FUNCTION_BLOCK FB_WATCHDOG_T (* Enables watchdog timeouts longer than the default. *)
  (* Standard: 61499-2; Description: TIMEOUT must be less than 15 s. The lower DT, the more accurate, but the higher the internal clock rate. *)
  (* Version 1.0, 2017-09-12, Marc Jakobi, HTW Berlin *)
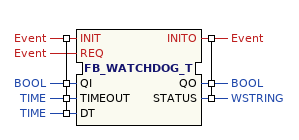
  EVENT_INPUT
    INIT WITH QI, TIMEOUT, DT; (* Initialization Request *)
    REQ; (* Normal Execution Request *)
  END_EVENT
  EVENT_OUTPUT
    INITO WITH QO, STATUS; (* Initialization Confirm *)
  END_EVENT
  VAR_INPUT
    QI : BOOL; (* Input event qualifier *)
    TIMEOUT : TIME; (* Watchdog timeout *)
    DT : TIME; (* Watchdog pet interval *)
  END_VAR
  VAR_OUTPUT
    QO : BOOL; (* Output event qualifier *)
    STATUS : WSTRING; (* Service status *)
  END_VAR
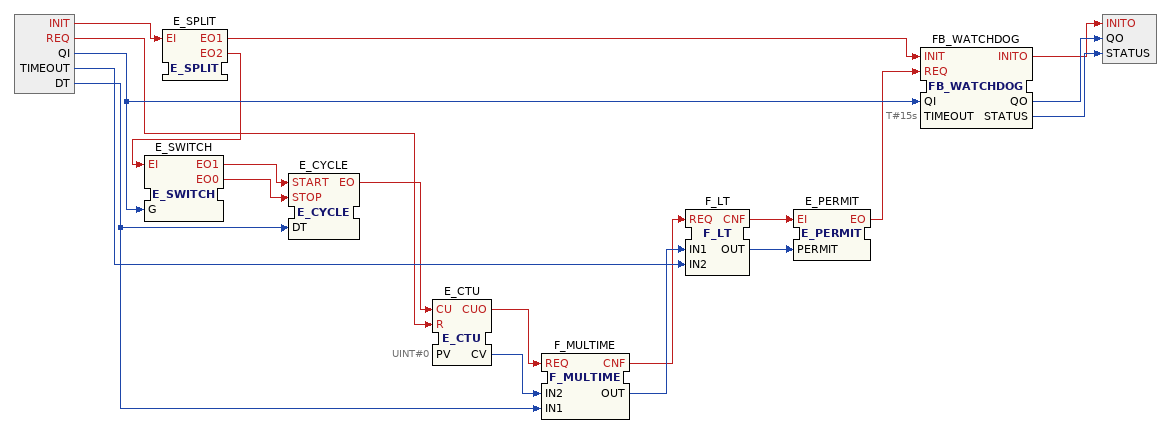
  FBS
    FB_WATCHDOG : FB_WATCHDOG(TIMEOUT := T#15s);
    E_CYCLE : E_CYCLE;
    E_SPLIT : E_SPLIT;
    E_SWITCH : E_SWITCH;
    E_CTU : E_CTU(PV := UINT#0);
    F_MULTIME : F_MULTIME;
    E_PERMIT : E_PERMIT;
    F_LT : F_LT;
  END_FBS
  EVENT_CONNECTIONS
    INIT TO E_SPLIT.EI;
    E_SPLIT.EO1 TO FB_WATCHDOG.INIT;
    E_SPLIT.EO2 TO E_SWITCH.EI;
    E_SWITCH.EO1 TO E_CYCLE.START;
    E_SWITCH.EO0 TO E_CYCLE.STOP;
    E_CYCLE.EO TO E_CTU.CU;
    REQ TO E_CTU.R;
    E_CTU.CUO TO F_MULTIME.REQ;
    F_MULTIME.CNF TO F_LT.REQ;
    F_LT.CNF TO E_PERMIT.EI;
    E_PERMIT.EO TO FB_WATCHDOG.REQ;
    FB_WATCHDOG.INITO TO INITO;
  END_CONNECTIONS
  DATA_CONNECTIONS
    QI TO FB_WATCHDOG.QI;
    QI TO E_SWITCH.G;
    DT TO E_CYCLE.DT;
    E_CTU.CV TO F_MULTIME.IN2;
    DT TO F_MULTIME.IN1;
    F_MULTIME.OUT TO F_LT.IN1;
    TIMEOUT TO F_LT.IN2;
    F_LT.OUT TO E_PERMIT.PERMIT;
    FB_WATCHDOG.QO TO QO;
    FB_WATCHDOG.STATUS TO STATUS;
  END_CONNECTIONS
END_FUNCTION_BLOCK
